TYPE AxisBeckhoff_t EXTENDS AxisBase_t :
STRUCT
    axis : AXIS_REF; // reference of the axis 
END_STRUCT
END_TYPE

(* stored: Version 1.1.0.1, ProductVersion 3.1.4024.6
   DUT AxisBeckhoff_t: Id {6fda199b-b00f-4961-846e-53893f7d0ce4} *)
